Universal Robots PolyScope program: ChamferFace.urp

Program ChamferFace (installation=main2 directory=/programs createdIn=5.11.5.1010327 lastSavedIn=5.11.5.1010327 robotSerialNumber=20215500677)
Calibrated DH parameters: a=[0.000204, -0.239222, -0.391845, -0.000001, 0.000022, 0]; d=[0.162722, -355.808559, 353.37206, 2.570385, 0.099741, 0.099629]; alpha=[1.571124, 0.000988, 0.008295, 1.568963, -1.570303, 0]; deltaTheta=[0, -0.973091, 7.204745, 0.05153, 0, 0]
Robot Program (runOnlyOnce=true)
  MoveJ speed 60 deg/s, acceleration 80 deg/s^2 (useActiveTCP=true) feature=Base
    Waypoint Waypoint_1: TCP in base x=52.074 y=-580.635 z=763.324 mm, rx=-0.4448 ry=1.1333 rz=-2.8534 rad; joints [69.674, -87.84, 62.052, 24.915, 60.899, -193.76] deg; TCP offset x=-1.34 y=-107.472 z=94.069 mm, rx=0.7854 ry=0 rz=0 rad
  MoveL speed 250 mm/s, acceleration 1200 mm/s^2 (useActiveTCP=true) feature=Base
    Waypoint Waypoint_2: TCP in base x=-350.229 y=-532.732 z=765.619 mm, rx=-0.2655 ry=-0.8484 rz=2.9475 rad; joints [33.921, -81.296, 61.468, 1.398, 43.388, -157.482] deg
